KUKA KRL program: inicializacion.src

&ACCESS RVP1
&REL 48
&PARAM TEMPLATE = C:\KRC\Roboter\Template\vorgabe
&PARAM EDITMASK = *
DEF inicializacion( )


;INICIALIZACION

CONTADOR_SACOS_darsena1=0
CONTADOR_CAPAS_darsena1=0
CAPA_ACTUAL_darsena1=0

CONTADOR_SACOS_darsena2=0
CONTADOR_CAPAS_darsena2=0
CAPA_ACTUAL_darsena2=0


LIMITE_CAPAS_DARSENA1=FALSE
LIMITE_CAPAS_DARSENA2=FALSE

END
